SUBAPPLICATION AX_SoftkeyToggle_RS_TO_QXA_BG (* Wraps AX_SoftkeyToggle_RS_TO_AX (Toggle/Reset-Zustand: SoftKey ODER AUX ODER lokale Web-/Dashboard-Methode ODER IO-Diag-Testbutton fuer den Toggle, SoftKey ODER AUX ODER Methode fuer den Reset) und treibt daraus 1 physischen Ausgang + Hintergrundfarbe (SoftKey+AUX-Handle+IO-Diag-Testbutton gemeinsam aus 1 GreenWhiteBackground4_AX) + lokalen State-Publish fuer Web-Client/OPC-Dashboard-Hintergrundfarbe. Generisch fuer jeden Ein/Aus-Ausgang, der von einer globalen Sammel-AUS-Taste mit-resettet werden muss (z.B. Saegeblattantrieb). *)
  (* Standard: 61499-2; Description: Copyright (c) 2026 Meisterschulen am Ostbahnhof This program and the accompanying materials are made available under the terms of the Eclipse Public License 2.0 which is available at https://www.eclipse.org/legal/epl-2.0/ SPDX-License-Identifier: EPL-2.0 *)
  (* Version 8.0, 2026-09-15, Franz Höpfinger, Meisterschulen am Ostbahnhof, FORCE_OFF Socket (AX) ergaenzt - reiner Durchreich-Socket an ToggleState.FORCE_OFF (AX_SoftkeyToggle_RS_TO_AX v1.2), analog AX_SoftkeyToggle_RS_TO_AX_BG_PUBLISH v1.1. Rein additiv, bestehende Instanzen muessen den neuen Socket verdrahten (z.B. auf einen festen FALSE-Literal, wenn nicht gebraucht). *)
  (* Version 7.0, 2026-09-12, Franz Höpfinger, Meisterschulen am Ostbahnhof, Toggle+Reset+AX_T_FF_SR nach MyLib::sys::AX_SoftkeyToggle_RS_TO_AX ausgelagert (Basis fuer Baender-Mehrkanal-Sequenzierung, die denselben Toggle/Reset-Unterbau braucht, aber mehrere zeitversetzte Ausgaenge statt 1). Diese SubApp ist jetzt nur noch der Wrapper: AX_SoftkeyToggle_RS_TO_AX + Ausgang/Hintergrund/Publish. Schnittstelle unveraendert. *)
  (* Version 6.0, 2026-09-11, Franz Höpfinger, Meisterschulen am Ostbahnhof, GreenWhiteBackground1_AX (2x, SoftKey allein + Testbutton allein) war falsch - ignorierte u16ObjIdA (AuxFunction2), Joystick-Handle bekam nie eine Rueckmeldung. Ersetzt durch 1 GreenWhiteBackground4_AX (SoftKey+AUX+Testbutton gemeinsam aus 1 Farbauswahl). AX_SPLIT_4 dadurch auf AX_SPLIT_3 verkleinert (nur noch logiBUS_QXA/Background/PUBLISH_STATE als Verbraucher). *)
  (* Version 5.0, 2026-09-11, Franz Höpfinger, Meisterschulen am Ostbahnhof, Softkey_Aux_Method_IE + Button_IE (Toggle-Zweig) kam als eigenes FB-Paar vor - nach MyLib::sys::Softkey_Aux_Method_Button_IE ausgelagert, 1 Instanz statt Sub-App+FB+2 EventConnections. u16ObjId_TEST bleibt zusaetzlich hier fuer die Hintergrundfarbe verdrahtet. Schnittstelle unveraendert. *)
  (* Version 4.0, 2026-09-11, Franz Höpfinger, Meisterschulen am Ostbahnhof, Softkey_Aux_IE + SERVER_0(+RSP) kam 2x vor (Toggle, Reset) - nach MyLib::sys::Softkey_Aux_Method_IE ausgelagert, je 1 Instanz statt 2 separater FB-Paare. Schnittstelle unveraendert. *)
  (* Version 3.0, 2026-09-11, Franz Höpfinger, Meisterschulen am Ostbahnhof, AUX (Joystick) ergaenzt - Toggle- und Reset-Softkey liefen durch MyLib::sys::Softkey_Aux_IE (SoftKey ODER AuxFunction2 -> 1 Event), statt den physischen Softkey allein per Softkey_IE zu lesen. Neue InputVars u16ObjIdA/u16ObjIdA_RESET (AuxFunction2_Saege_EinAus/AuxFunction2_AUS fuer den Saege-Anwendungsfall). Wechselt Trigger-Moment des Softkeys von SK_RELEASED auf SK_PRESSED (Softkey_Aux_IE-Konvention, einzig sinnvolle 'aktiviert'-Bedeutung fuer eine Merge-Anwendung mit AUX). *)
  (* Version 2.0, 2026-09-11, Franz Höpfinger, Meisterschulen am Ostbahnhof, IO-Diag-Testbutton (u16ObjId_TEST) und 2 lokale RPC-Methoden (ID_TOGGLE_METHOD/ID_RESET_METHOD) + State-Publish (ID_STATE_WRITE) ergaenzt, damit IO-Diag-Screen UND Web-Client/OPC-Dashboard gleichberechtigt am selben AX_T_FF_SR haengen statt am (bisher orphanten) rohen Testbutton bzw. gar nicht (Web). *)
  (* Version 1.0, 2026-09-11, Franz Höpfinger, Meisterschulen am Ostbahnhof, initial implementation - Reset-Set-Toggle-Variante von AX_SoftkeyToggle_TO_QXA_BG (AX_T_FF statt AX_T_FF_SR), fuer Ausgaenge mit zusaetzlicher globaler AUS-Taste (Saegeblattantrieb: SoftKey_Saege_EinAus toggelt, SoftKey_AUS resettet). *)
  PACKAGE MyLib::sys;
  IMPORT isobus::UT::Q::const::IDs::ID_NULL;
  IMPORT logiBUS::io::DQ::logiBUS_DO;
  IMPORT logiBUS::io::DQ::logiBUS_DO_S;
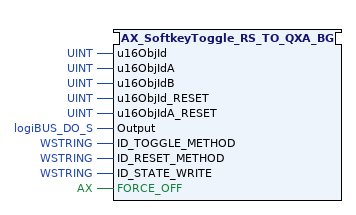
  VAR_INPUT
    u16ObjId : UINT := ID_NULL; (* Object ID Softkey Ein/Aus (Toggle), traegt auch die Hintergrundfarbe *)
    u16ObjIdA : UINT := ID_NULL; (* Object ID AuxFunction2 (Joystick) fuer den Toggle - gleichberechtigt zum SoftKey, zeigt Hintergrundfarbe am Aux-Handle mit *)
    u16ObjIdB : UINT := ID_NULL; (* Object ID IO-Diag-Testbutton (Ausgaenge-Diagnoseseite) - toggelt gleichberechtigt mit, zeigt Hintergrundfarbe gemeinsam mit SoftKey+AUX *)
    u16ObjId_RESET : UINT := ID_NULL; (* Object ID Softkey 'Alles Aus' (Reset, hart auf AUS) - z.B. SoftKey_AUS *)
    u16ObjIdA_RESET : UINT := ID_NULL; (* Object ID AuxFunction2 (Joystick) fuer den Reset - gleichberechtigt zum Softkey 'Alles Aus' *)
    Output : logiBUS::io::DQ::logiBUS_DO_S := logiBUS_DO::Invalid; (* Identify the Output Output_Q1..Q12 *)
    ID_TOGGLE_METHOD : WSTRING; (* Lokale Methodenadresse (ACTION=CREATE_METHOD) fuer den argumentlosen Toggle-Trigger - wird von Web-Client (vt-ui-mirror) UND direkt vom OPC-Dashboard aufgerufen *)
    ID_RESET_METHOD : WSTRING; (* Lokale Methodenadresse (ACTION=CREATE_METHOD) fuer den argumentlosen Reset-Trigger (hart auf AUS) - wird von Web-Client UND OPC-Dashboard aufgerufen *)
    ID_STATE_WRITE : WSTRING; (* Lokale Publish-Adresse (ACTION=WRITE) fuer den tatsaechlichen Toggle-Zustand (AX_T_FF_SR.Q) - wird von Web-Client/Dashboard remote abonniert *)
  END_VAR
  SOCKETS
    FORCE_OFF : adapter::types::unidirectional::AX; (* Optional: steigende Flanke resettet hart auf AUS (z.B. Sicherheitsabschaltung) - reiner Durchreich-Socket an ToggleState.FORCE_OFF. Unverdrahtet lassen (fester FALSE-Literal), wenn nicht gebraucht. *)
  END_SOCKETS
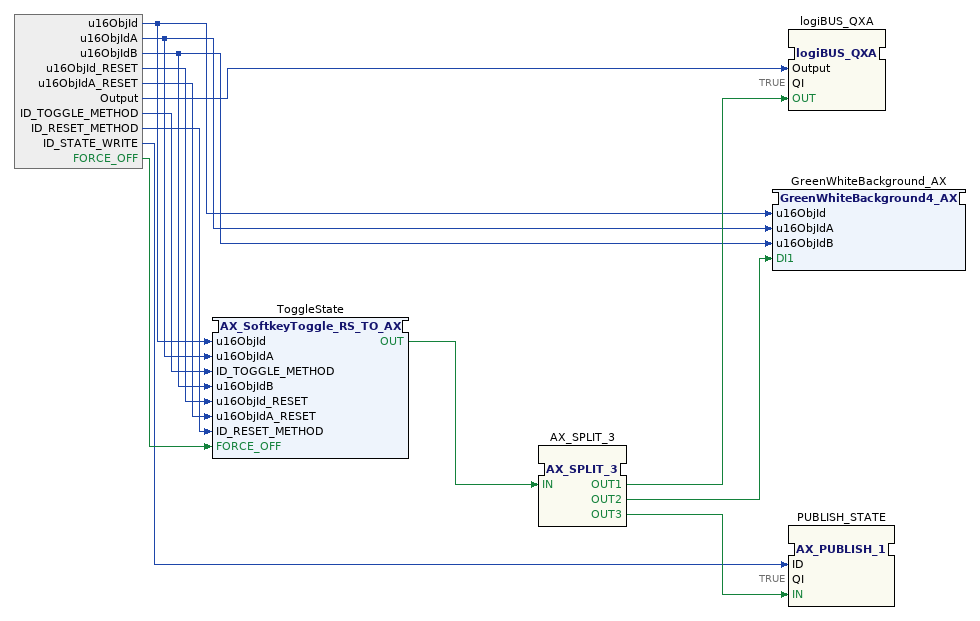
  FBS
    AX_SPLIT_3 : adapter::events::unidirectional::AX_SPLIT_3;
    logiBUS_QXA : logiBUS::io::DQ::logiBUS_QXA(QI := TRUE);
    PUBLISH_STATE : adapter::net::AX_PUBLISH_1(QI := TRUE);
  END_FBS
  SUBAPPS
    ToggleState : MyLib::sys::AX_SoftkeyToggle_RS_TO_AX;
    GreenWhiteBackground_AX : MyLib::sys::GreenWhiteBackground4_AX;
  END_SUBAPPS
  DATA_CONNECTIONS
    u16ObjId TO ToggleState.u16ObjId;
    u16ObjIdA TO ToggleState.u16ObjIdA;
    ID_TOGGLE_METHOD TO ToggleState.ID_TOGGLE_METHOD;
    u16ObjIdB TO ToggleState.u16ObjIdB;
    u16ObjId_RESET TO ToggleState.u16ObjId_RESET;
    u16ObjIdA_RESET TO ToggleState.u16ObjIdA_RESET;
    ID_RESET_METHOD TO ToggleState.ID_RESET_METHOD;
    u16ObjId TO GreenWhiteBackground_AX.u16ObjId;
    u16ObjIdA TO GreenWhiteBackground_AX.u16ObjIdA;
    u16ObjIdB TO GreenWhiteBackground_AX.u16ObjIdB;
    Output TO logiBUS_QXA.Output;
    ID_STATE_WRITE TO PUBLISH_STATE.ID;
  END_CONNECTIONS
  ADAPTER_CONNECTIONS
    ToggleState.OUT TO AX_SPLIT_3.IN;
    AX_SPLIT_3.OUT1 TO logiBUS_QXA.OUT;
    AX_SPLIT_3.OUT2 TO GreenWhiteBackground_AX.DI1;
    AX_SPLIT_3.OUT3 TO PUBLISH_STATE.IN;
    FORCE_OFF TO ToggleState.FORCE_OFF;
  END_CONNECTIONS
END_SUBAPPLICATION
